Staubli VAL3: ExtraSysAxisIni.pgx

public program ExtraSysAxisIni(bool& x_bRes)
begin

  //2014.07.28
  //同步七八轴

  x_bRes=false
  TxtFile:bSync7Axis=TxtFile:bSync8Axis=false
  if $fileExists("Usr://configs/externaxes.cfx") and getVersion("externalAxis")!="false"

    if !ExtAxis:libExist("Disk://extAxisCan/extAxisCan.pjx")

      //2014.08.06
      //适配7.5版本和S7.6版本
      if find(getVersion("System"),"s7.5")>=0
        if !$copy("Disk://extAxisCan/TASK4MS7.5.pgx","Disk://extAxisCan/TASK4MS.pgx")
          popUpMsg("外部轴TASK4MS程序不正确")
          return
        endIf

      else
        if !$copy("Disk://extAxisCan/TASK4MS7.6.pgx","Disk://extAxisCan/TASK4MS.pgx")
          popUpMsg("外部轴TASK4MS程序不正确")
          return
        endIf
      endIf

      //


      if ExtAxis:libLoad("Disk://extAxisCan/extAxisCan.pjx")!=0
        popUpMsg("加载同步轴库不正确")
        return
      endIf
    endIf
    call ExtAxis:CheckAxis(TxtFile:bSync7Axis,TxtFile:bSync8Axis)
    call ExtAxis:init()
    // call ExtAxis:Reset()
    DataBase:nAsysAxisPer=max(0.004,DataBase:nAsysAxisPer)
    taskCreateSync "SyncAxis",DataBase:nAsysAxisPer,bSync,ExtAxis:Task4ms()

  endIf

  x_bRes=true





end
